// TIA Portal V17 export
// export: Created 2025-06-26T07:49:34.9666636Z, ExportSetting WithDefaults, DisplayName Totally Integrated Automation Portal, DisplayVersion V17 Update 8, DisplayName TIA Portal Openness, DisplayVersion V17 Update 8, DisplayName TIA Portal Version Control Interface, DisplayVersion V17, DisplayName STEP 7 Professional, DisplayVersion V17 Update 8, DisplayName STEP 7 Safety, DisplayVersion V17 Update 6, DisplayName WinCC Advanced, DisplayVersion V17 Update 8
FUNCTION_BLOCK "Initialise"   // FB25, FBD
{ S7_Optimized_Access := 'TRUE' }
AUTHOR : Heaten
VERSION : 0.1
// stored: AutoNumber true, IsIECCheckEnabled false, IsRetainMemResEnabled false, MemoryReserve 0, SetENOAutomatically false, UDAEnableTagReadback false
   VAR_INPUT
      bEnable { ExternalAccessible := 'False'; ExternalVisible := 'False'; ExternalWritable := 'False'} : Bool;
      bOverwriteParameters { ExternalAccessible := 'False'; ExternalVisible := 'False'; ExternalWritable := 'False'} : Bool;   // Overwrite DB_CurrentSetting from DB_StaticData
   END_VAR
   VAR_OUTPUT
      Done { ExternalAccessible := 'False'; ExternalVisible := 'False'; ExternalWritable := 'False'} : Bool;
   END_VAR
   VAR
      "Step" { ExternalAccessible := 'False'; ExternalVisible := 'False'; ExternalWritable := 'False'} : Int;
      Step_0 { ExternalAccessible := 'False'; ExternalVisible := 'False'; ExternalWritable := 'False'} : Bool;
      Step_1 { ExternalAccessible := 'False'; ExternalVisible := 'False'; ExternalWritable := 'False'} : Bool;
      Step_2 { ExternalAccessible := 'False'; ExternalVisible := 'False'; ExternalWritable := 'False'} : Bool;
      Step_3 { ExternalAccessible := 'False'; ExternalVisible := 'False'; ExternalWritable := 'False'} : Bool;
      Step_4 { ExternalAccessible := 'False'; ExternalVisible := 'False'; ExternalWritable := 'False'} : Bool;
      RetVal_Fluid { ExternalAccessible := 'False'; ExternalVisible := 'False'; ExternalWritable := 'False'} : Word;   // Static for debug purposes
      RetVal_System { ExternalAccessible := 'False'; ExternalVisible := 'False'; ExternalWritable := 'False'} : Word;   // Static for debug purposes
      RetVal_Compressor { ExternalAccessible := 'False'; ExternalVisible := 'False'; ExternalWritable := 'False'} : Word;   // Static for debug purposes
      A0003 { ExternalAccessible := 'False'; ExternalVisible := 'False'; ExternalWritable := 'False'} : "fbHMIEvent";
   END_VAR
   VAR_TEMP
      Busy : Bool;
   END_VAR
   VAR_TEMP   // added for the SCL form of the ladder/FBD networks
      _w1 : Bool;
   END_VAR
BEGIN

REGION Network 1 (SCL): Initialize step control
   IF (#bEnable = TRUE OR #bOverwriteParameters = TRUE) AND #Step_0 = FALSE AND #Step_1 = FALSE AND #Step_2 = FALSE AND #Step_3 = FALSE AND #Step_4 = FALSE THEN
       #Step_0 := TRUE;
       #Done := False;
   END_IF;
END_REGION

REGION Network 2 (SCL): Step_0: Set basic settings
   IF #Step_0 THEN

       "DB_State".State."0_Initialisation" := TRUE;

       "DB_State".State."1_Offline" :=
       "DB_State".State."2_Standby" :=
       "DB_State".State."3_PrepareStart" :=
       "DB_State".State."4_Start" :=
       "DB_State".State."5_Warmup" :=
       "DB_State".State."6_Running" :=
       "DB_State".State."7_Stop" := FALSE;

       //"DB_Alarms"."0001_WatchdogTimeoutOB1".bActive := FALSE;

       // Temporarily set some settings here. This should be changeable by the user via RETAIN variables.

      // "DB_CurrentSetting".VariableSetting.SystemType := 6;            // 1 = Test Station, 2 = Only cabinet, 3 = Ant, 4 = Bee, 5 = Cicada, 6 = HB-L4 Alpha
      // "DB_CurrentSetting".VariableSetting.FluidType := 1;             // 1 = R245fa
      // "DB_CurrentSetting".VariableSetting.CompressorType := 1;        // 1 = 1st Generation
      // "DB_CurrentSetting".VariableSetting.InstalledCompressors[8] := TRUE;
      "DB_CurrentSetting".VariableSetting.EnableViaHMI := TRUE;
       //"DB_Regulators".PerformanceControl.Settings.HeatSink.HeatSinkTemperatureControl_Active := TRUE;
       //"DB_Regulators".PerformanceControl.Settings.HeatSource.HeatSourceTemperatureControl_Active := FALSE;
       //"DB_Regulators".PerformanceControl.Settings.VariableControl.Control_Active := FALSE;

       //"DB_CurrentSetting".VariableSetting.ActiveCompressors := "DB_CurrentSetting".VariableSetting.InstalledCompressors;


       #Step_0 := FALSE;
       #Step_1 := TRUE;

   END_IF;
END_REGION

REGION Network 3 (SCL): Step_1: Currently not used

   IF #Step_1 THEN
       (* anything to do here? *)
       #Step_1 := FALSE;
       #Step_2 := TRUE;
   END_IF;
END_REGION

REGION Network 4: Step_2: Overwrite parameters
   // Load settings from Static DB if requested
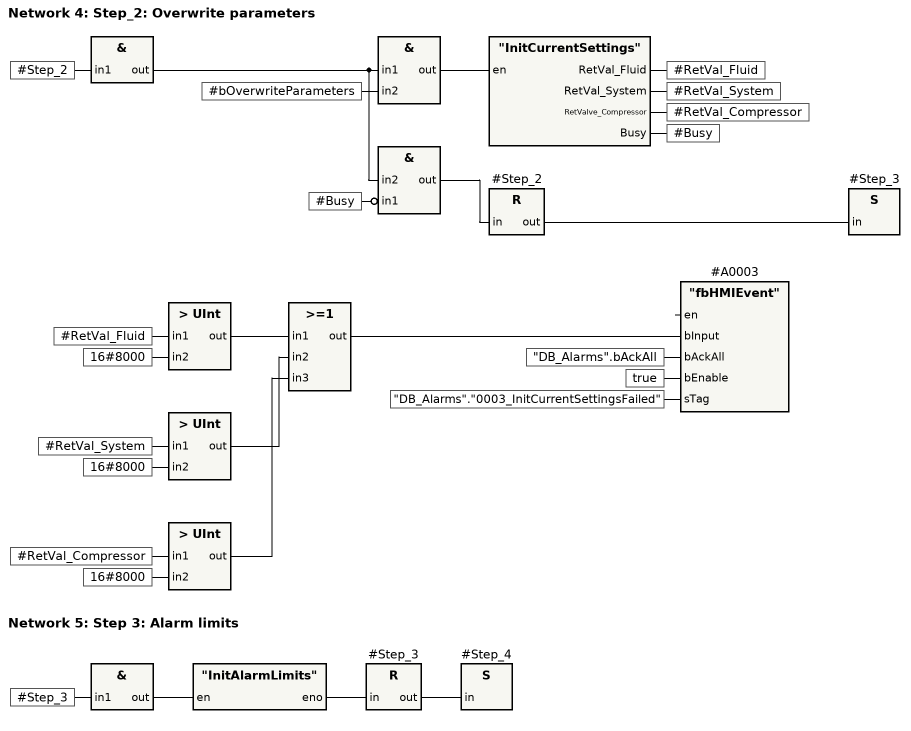
   IF #Step_2 AND #bOverwriteParameters THEN
       "InitCurrentSettings"(RetVal_Fluid => #RetVal_Fluid,
                             RetVal_System => #RetVal_System,
                             RetValve_Compressor => #RetVal_Compressor,
                             Busy => #Busy);
   END_IF;
   #_w1 := #Step_2 AND NOT #Busy;
   IF #_w1 THEN
       #Step_2 := FALSE;
       #Step_3 := TRUE;
   END_IF;
   #A0003(bInput := (#RetVal_Fluid > 16#8000) OR (#RetVal_System > 16#8000) OR (#RetVal_Compressor > 16#8000),   // "fbHMIEvent"
          bAckAll := "DB_Alarms".bAckAll,
          bEnable := true,
          sTag := "DB_Alarms"."0003_InitCurrentSettingsFailed");
END_REGION

REGION Network 5: Step 3: Alarm limits
   "InitAlarmLimits"(EN := #Step_3, ENO => #_w1);
   IF #_w1 THEN
       #Step_3 := FALSE;
       #Step_4 := TRUE;
   END_IF;
END_REGION

REGION Network 6 (SCL): Step 4
   IF #Step_4 THEN
       "DB_CurrentSetting".ParameterSet_Ordered := False;
       #Step_4 := FALSE;
       "DB_Alarms".bAckAll := TRUE; 
       #Done := True;
   END_IF;
END_REGION
END_FUNCTION_BLOCK
